FUNCTION_BLOCK CfbBreakerController
  (* Standard: 61499-2 *)
  (* Version 0.1, 2019-00-29, hpea485, UOA *)
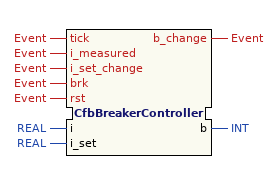
  EVENT_INPUT
    tick;
    i_measured;
    i_set_change;
    brk;
    rst;
  END_EVENT
  EVENT_OUTPUT
    b_change;
  END_EVENT
  VAR_INPUT
    i : REAL;
    i_set : REAL;
  END_VAR
  VAR_OUTPUT
    b : INT;
  END_VAR
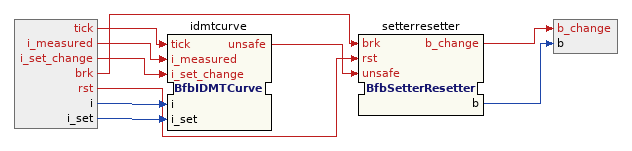
  FBS
    idmtcurve : BfbIDMTCurve;
    setterresetter : BfbSetterResetter;
  END_FBS
  EVENT_CONNECTIONS
    tick TO idmtcurve.tick;
    i_measured TO idmtcurve.i_measured;
    i_set_change TO idmtcurve.i_set_change;
    brk TO setterresetter.brk;
    rst TO setterresetter.rst;
    setterresetter.b_change TO b_change;
    idmtcurve.unsafe TO setterresetter.unsafe;
  END_CONNECTIONS
  DATA_CONNECTIONS
    i TO idmtcurve.i;
    i_set TO idmtcurve.i_set;
    setterresetter.b TO b;
  END_CONNECTIONS
END_FUNCTION_BLOCK
